FUNCTION_BLOCK AutomaticFlowControlHandler
VAR_OUTPUT
	controlValvePercentage : INT;
END_VAR
VAR
END_VAR

END_FUNCTION_BLOCK

(* stored: Version 1.1.0.1, ProductVersion 3.1.4024.9
   POU AutomaticFlowControlHandler: Id {1d683a84-77f3-4fa0-9fcb-6c948632e209}, SpecialFunc None *)
